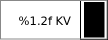
VISUALIZATION VISU_ALIM_HT_S10  // 108x40
VAR_IN_OUT
	m_Input_HT:				BLOCK_CANON_ST10;
END_VAR
VAR_IN_OUT
END_VAR
    Rectangle (84,2 20x35), colour toggle: m_Input_HT.STATE_HV_ON, invisible if: NOT m_Input_HT.STATE_HV_ON AND NOT m_Input_HT.STATE_HV
    Rectangle (84,2 20x35), invisible if: m_Input_HT.STATE_HV_ON OR m_Input_HT.STATE_HV
    Polygon (41,73)
    Rectangle (80,0 28x40), invisible if: NOT m_Input_HT.HV.AUTOR_On_IHM AND NOT m_Input_HT.HV.AUTOR_Off_IHM, input disabled if: (NOT m_Input_HT.HV.AUTOR_ON_IHM AND NOT m_Input_HT.HV.AUTOR_OFF_IHM) OR NOT PRG_User.ACTU_USER.MAINTENANCE
        tap m_Input_HT.HV.M_On
    Rectangle (11,15 71x12), "%1.2f KV", text variable: m_Input_HT.STATE_V_HV
END_VISUALIZATION

(* stored: Version 1.1.0.1, ProductVersion 3.1.4024.10
   Visu VISU_ALIM_HT_S10: Id {6be1f3ff-6c8e-47b8-9cea-3942a5d37e08} *)
